{attribute 'to_string'}
TYPE TReadSymbolTableState :
(
	RS_WAIT_FOR_START,
	RS_READ_SYMBOL_UPLOAD_INFO,
	RS_READ_SYMBOL_UPLOAD,
	RS_PROCESS_SYMBOL_UPLOAD,
	RS_DONE
	
);
END_TYPE

(* stored: Version 1.1.0.1, ProductVersion 3.1.4024.3
   DUT TReadSymbolTableState: Id {161c7e9b-c20e-48cc-a5e1-e506835a0204} *)
